Staubli VAL3: SAVEtoolAfranme.pgx

program SAVEtoolAfranme()
begin
  for nframe=0 to 9
    lib:frmaster[nframe].trsf=frmaster[nframeSave[nframe]].trsf
  endFor
  for ntool=0 to 9
    lib:t2[ntool].trsf=t2[ntoolSave[ntool]].trsf
  endFor
end
